INTERFACE I_LinkedListNode EXTENDS I_Disposable

PROPERTY PUBLIC DataSize : UDINT
GET
END_GET
END_PROPERTY

METHOD PUBLIC Equals : BOOL
VAR_INPUT
	Symbol : ANY;
END_VAR
END_METHOD

METHOD PUBLIC Get : BOOL;
VAR_INPUT
	Destination : ANY;
END_VAR
END_METHOD

METHOD PUBLIC GetTo : BOOL;
VAR_INPUT
	Destination : PVOID;
	DestinationSize : UDINT;
END_VAR
END_METHOD

PROPERTY PUBLIC Next : I_LinkedListNode
GET
END_GET
SET
END_SET
END_PROPERTY

PROPERTY PUBLIC Previous : I_LinkedListNode
GET
END_GET
SET
END_SET
END_PROPERTY

END_INTERFACE

(* stored: Version 1.1.0.1, ProductVersion 3.1.4024.12
   Itf I_LinkedListNode: Id {947b0a6f-b18c-4037-bae0-12d338be00da}
   Property DataSize: Id {18f9a4c9-70bc-4e4c-9f32-d840e79da13f}
   Get Get: Id {cfeb2235-325a-4950-ac6e-b849773697df}
   Method Equals: Id {a343db1e-bd0d-40a4-b217-2c35870d68a4}
   Method Get: Id {e3aaadc9-a69b-4db5-8f6e-b807b798613c}
   Method GetTo: Id {b3c69cd4-1eac-4cd3-a874-6b8d5dc47719}
   Property Next: Id {04648973-8c2a-4589-8746-2a0ee739b1fb}
   Get Get: Id {1478ef3b-5f53-42fe-ab3e-ac8a03c19848}
   Set Set: Id {23c6723b-f3c5-4a63-8385-34ae4ca393b5}
   Property Previous: Id {317c7db0-7c68-4af7-b234-bd49ca7cb32d}
   Get Get: Id {18784a87-ec8d-4104-83b6-770e64bdeb1b}
   Set Set: Id {30518ff6-4f33-4bcc-bc11-97685f488e23} *)
